AssertEquals(
    Expected := expected,
    Actual := actual,
    Message := 'Value did not update target'
);

TEST_FINISHED();
END_METHOD

METHOD PUBLIC TestSerializeTypeWith
VAR
    _type : _LINT(0);
    serializer : JsonSerializer;
    expected : STRING(500) := '{"typeName":"LINT","minValue":-9223372036854775808,"maxValue":9223372036854775807,"isSigned":true,"isFloat":false}';
    actual : STRING(500);
END_VAR
TEST('TestSerializeTypeWith');

serializer.Reset();
_type.SerializeTypeWith(serializer);
serializer.TryGetSerializedData(ADR(actual), SIZEOF(actual));

AssertEquals_STRING(
    Expected := expected,
    Actual := actual,
    Message := 'Serialization of type did not return correct string.'
);

TEST_FINISHED();
END_METHOD

METHOD PUBLIC TestSerializeWith
VAR
    _type : _LINT(32767);
    serializer : JsonSerializer;
    expected : STRING := '32767';
    actual : STRING(500);
END_VAR
TEST('TestSerializeWith');

serializer.Reset();
_type.SerializeWith(serializer);
serializer.TryGetSerializedData(ADR(actual), SIZEOF(actual));

AssertEquals_STRING(
    Expected := expected,
    Actual := actual,
    Message := 'Serialization of type data did not return correct string.'
);

TEST_FINISHED();
END_METHOD

METHOD PUBLIC TestSize
VAR
    _type : _LINT(0);
    expected : UDINT := SIZEOF(LINT);
    actual : UDINT;
END_VAR
TEST('TestSize');

actual := _type.Size;

AssertEquals_UDINT(
    Expected := Expected,
    Actual := actual,
    Message := 'Type did not return the correct size.'
);

TEST_FINISHED();
END_METHOD

METHOD PUBLIC TestTryDeserializeFrom
VAR
    deserializer : JsonDeserializer;
    feedback : DeserializerFeedback;
    json : STRING := '32767';
    _type : _LINT(0);
    expected : LINT := 32767;
    actual : LINT;
 END_VAR
TEST('TestTryDeserializeFrom');

deserializer.Reset();
deserializer.TryLoad(json);
_type.TryDeserializeFrom(Deserializer, Feedback);

actual := _type.Value;

AssertEquals(
    Expected := expected,
    Actual := actual,
    Message := 'Type did not deserialize correctly.'
);

TEST_FINISHED();
END_METHOD

METHOD PUBLIC TestTryMakeReferenceToFollowsReference
VAR
    _type : _LINT(0);
	target : _LINT(0);
    expected : LINT := 123;
    actual : LINT;
END_VAR
TEST('TestTryMakeReferenceToFollowsReference');

_type.TryMakeReferenceTo(target);
target.Value := 123;

actual := _type.Value;

AssertEquals(
    Expected := expected,
    Actual := actual,
    Message := 'Value did not follow target change'
);

TEST_FINISHED();
END_METHOD

METHOD PUBLIC TestTryMakeReferenceToUpdatesReference
VAR
    _type : _LINT(0);
	target : _LINT(0);
    expected : LINT := 123;
    actual : LINT;
END_VAR
TEST('TestTryMakeReferenceToUpdatesReference');

_type.TryMakeReferenceTo(target);
_type.Value := 123;

actual := target.Value;

AssertEquals(
    Expected := expected,
    Actual := actual,
    Message := 'Value did not update target'
);

TEST_FINISHED();
END_METHOD

METHOD PUBLIC TestTypeNameReturnsExpected
VAR
    _type : _LINT(0);
    expected : STRING := 'LINT';
    actual : STRING;
END_VAR
TEST('TestTypeNameReturnsExpected');

actual := _type.TypeName;

AssertEquals_STRING(
    Expected := expected,
    Actual := actual,
    Message := 'Type did not return correct iec type.'
);

TEST_FINISHED();
END_METHOD

METHOD PUBLIC TestValueReturnsExpectedAfterChange
VAR
    _type : _LINT(0);
    expected : LINT := 32767;
    actual : LINT;
END_VAR
TEST('TestValueReturnsExpectedAfterChange');

_type.Value := 32767;

actual := _type.Value;

AssertEquals(
    Expected := expected,
    Actual := actual,
    Message := 'Expected value not returned after change.'
);

TEST_FINISHED();
END_METHOD

METHOD PUBLIC TestValueReturnsExpectedAfterInit
VAR
    _type : _LINT(32767);
    expected : LINT := 32767;
    actual : LINT;
END_VAR
TEST('TestValueReturnsExpectedAfterInit');

actual := _type.Value;

AssertEquals(
    Expected := expected,
    Actual := actual,
    Message := 'Expected value not returned after Init.'
);

TEST_FINISHED();
END_METHOD

END_FUNCTION_BLOCK

// ---- mobject-datatypes/Tests/_REAL_TestSuite.TcPOU
FUNCTION_BLOCK _REAL_TestSuite EXTENDS TcUnit.FB_TestSuite
VAR
END_VAR

TestAddress();
TestClearReference();
TestClone();
TestTypeNameReturnsExpected();
TestIsFloat();
TestIsSigned();
TestMakeReferenceToFollowsReference();
TestMakeReferenceToUpdatesReference();
TestSize();
TestValueReturnsExpectedAfterInit();
TestValueReturnsExpectedAfterChange();
TestSerializeTypeWith();
TestSerializeWith();
TestTryDeserializeFrom();
TestTryMakeReferenceToFollowsReference();
TestTryMakeReferenceToUpdatesReference();

METHOD PUBLIC TestAddress
VAR
    _type : _REAL(0.0);
    notExpected : PVOID := 0;
    actual : PVOID;
END_VAR
TEST('TestAddress');

actual := _type.Address;

AssertFalse(
    Condition := (notExpected = actual),
    Message := 'Type did not return a valid address.'
);

TEST_FINISHED();
END_METHOD

METHOD PUBLIC TestClearReference
VAR
    _type : _REAL(0.0);
	target : REAL := 0.0;
    expected : REAL := 0.0;
    actual : REAL;
END_VAR
TEST('TestClearReference');

_type.MakeReferenceTo(target);
_type.ClearReference();
target := 123.4;

actual := _type.Value;

AssertEquals_REAL(
    Expected := expected,
    Actual := actual,
    Delta := REAL#0.001,
    Message := 'Value incorrectly followed target change'
);

TEST_FINISHED();
END_METHOD

METHOD PUBLIC TestClone
VAR
    _type : _REAL(123.4);
	clone : I_Datatype;
	isValidClone : BOOL;
	compareResult : DINT;
END_VAR
TEST('TestClone');

clone := _type.Clone();

isValidClone := clone <> 0;

IF isValidClone THEN
	compareResult := memcmp(_type.Address, clone.Address, clone.Size);
END_IF

AssertTrue(
	Condition := isValidClone,
	Message := 'Clone did not produce a clone'
);

AssertEquals_DINT(
	Expected := 0,
    Actual := compareResult,
    Message := 'Clone did not return a valid clone.'
);

clone.Dispose();

TEST_FINISHED();
END_METHOD

METHOD PUBLIC TestIsFloat
VAR
    _type : _REAL(0);
END_VAR
TEST('TestIsFloat');

AssertTrue(
	Condition := _type.IsFloat,
    Message := 'Type did not correctly identify itself as being unsigned'
);

TEST_FINISHED();
END_METHOD

METHOD PUBLIC TestIsSigned
VAR
    _type : _REAL(0);
END_VAR
TEST('TestIsSigned');

AssertTrue(
	Condition := _type.IsSigned,
    Message := 'Type did not correctly identify itself as being signed'
);

TEST_FINISHED();
END_METHOD

METHOD PUBLIC TestMakeReferenceToFollowsReference
VAR
    _type : _REAL(0.0);
	target : REAL := 0.0;
    expected : REAL := 123.4;
    actual : REAL;
END_VAR
TEST('TestMakeReferenceToFollowsReference');

_type.MakeReferenceTo(target);
target := 123.4;

actual := _type.Value;

AssertEquals_REAL(
    Expected := expected,
    Actual := actual,
    Delta := REAL#0.001,
    Message := 'Value did not follow target change'
);

TEST_FINISHED();
END_METHOD

METHOD PUBLIC TestMakeReferenceToUpdatesReference
VAR
    _type : _REAL(0.0);
	target : REAL := 0.0;
    expected : REAL := 123.4;
    actual : REAL;
END_VAR
TEST('TestMakeReferenceToUpdatesReference');

_type.MakeReferenceTo(target);
_type.Value := 123.4;

actual := target;

AssertEquals_REAL(
    Expected := expected,
    Actual := actual,
    Delta := REAL#0.001,
    Message := 'Value did not update target'
);

TEST_FINISHED();
END_METHOD

METHOD PUBLIC TestSerializeTypeWith
VAR
    _type : _REAL(0.0);
    serializer : JsonSerializer;
    expected : STRING(500) := '{"typeName":"REAL","minValue":-3.4028230607370965e38,"maxValue":3.4028230607370965e38,"isSigned":true,"isFloat":true}';
    actual : STRING(500);
END_VAR
TEST('TestSerializeTypeWith');

serializer.Reset();
_type.SerializeTypeWith(serializer);
serializer.TryGetSerializedData(ADR(actual), SIZEOF(actual));

AssertEquals_STRING(
    Expected := expected,
    Actual := actual,
    Message := 'Serialization of type did not return correct string.'
);

TEST_FINISHED();
END_METHOD

METHOD PUBLIC TestSerializeWith
VAR
    _type : _REAL(123.4);
    serializer : JsonSerializer;
    expected : STRING := '123.4000015258789'; // Expected value due to the nature of floating point values defined by IEEE754.
    actual : STRING(500);
END_VAR
TEST('TestSerializeWith');

serializer.Reset();
_type.SerializeWith(serializer);
serializer.TryGetSerializedData(ADR(actual), SIZEOF(actual));

AssertEquals_STRING(
    Expected := expected,
    Actual := actual,
    Message := 'Serialization of type data did not return correct string.'
);

TEST_FINISHED();
END_METHOD

METHOD PUBLIC TestSize
VAR
    _type : _REAL(0.0);
    expected : UDINT := SIZEOF(REAL);
    actual : UDINT;
END_VAR
TEST('TestSize');

actual := _type.Size;

AssertEquals_UDINT(
    Expected := Expected,
    Actual := actual,
    Message := 'Type did not return the correct size.'
);

TEST_FINISHED();
END_METHOD

METHOD PUBLIC TestTryDeserializeFrom
VAR
    deserializer : JsonDeserializer;
    feedback : DeserializerFeedback;
    json : STRING := '123.4';
    _type : _REAL(0.0);
    expected : REAL := 123.4;
    actual : REAL;
 END_VAR
TEST('TestTryDeserializeFrom');

deserializer.Reset();
deserializer.TryLoad(json);
_type.TryDeserializeFrom(Deserializer, Feedback);

actual := _type.Value;

AssertEquals_REAL(
    Expected := expected,
    Actual := actual,
    Delta := REAL#0.001,
    Message := 'Type did not deserialize correctly.'
);

TEST_FINISHED();
END_METHOD

METHOD PUBLIC TestTryMakeReferenceToFollowsReference
VAR
    _type : _REAL(0.0);
	target : _REAL(0.0);
    expected : REAL := 123.4;
    actual : REAL;
END_VAR
TEST('TestTryMakeReferenceToFollowsReference');

_type.TryMakeReferenceTo(target);
target.Value := 123.4;

actual := _type.Value;

AssertEquals_REAL(
    Expected := expected,
    Actual := actual,
    Delta := REAL#0.001,
    Message := 'Value did not follow target change'
);

TEST_FINISHED();
END_METHOD

METHOD PUBLIC TestTryMakeReferenceToUpdatesReference
VAR
    _type : _REAL(0.0);
	target : _REAL(0.0);
    expected : REAL := 123.4;
    actual : REAL;
END_VAR
TEST('TestTryMakeReferenceToUpdatesReference');

_type.TryMakeReferenceTo(target);
_type.Value := 123.4;

actual := target.Value;

AssertEquals_REAL(
    Expected := expected,
    Actual := actual,
    Delta := REAL#0.001,
    Message := 'Value did not update target'
);

TEST_FINISHED();
END_METHOD

METHOD PUBLIC TestTypeNameReturnsExpected
VAR
    _type : _REAL(0.0);
    expected : STRING := 'REAL';
    actual : STRING;
END_VAR
TEST('TestTypeNameReturnsExpected');

actual := _type.TypeName;

AssertEquals_STRING(
    Expected := expected,
    Actual := actual,
    Message := 'Type did not return correct iec type.'
);

TEST_FINISHED();
END_METHOD

METHOD PUBLIC TestValueReturnsExpectedAfterChange
VAR
    _type : _REAL(0.0);
    expected : REAL := 123.4;
    actual : REAL;
END_VAR
TEST('TestValueReturnsExpectedAfterChange');

_type.Value := 123.4;

actual := _type.Value;

AssertEquals_REAL(
    Expected := expected,
    Actual := actual,
    Delta := REAL#0.001,
    Message := 'Expected value not returned after change.'
);

TEST_FINISHED();
END_METHOD

METHOD PUBLIC TestValueReturnsExpectedAfterInit
VAR
    _type : _REAL(123.4);
    expected : REAL := 123.4;
    actual : REAL;
END_VAR
TEST('TestValueReturnsExpectedAfterInit');

actual := _type.Value;

AssertEquals_REAL(
    Expected := expected,
    Actual := actual,
    Delta := REAL#0.001,
    Message := 'Expected value not returned after Init.'
);

TEST_FINISHED();
END_METHOD

END_FUNCTION_BLOCK

// ---- mobject-datatypes/Tests/_SINT_TestSuite.TcPOU
FUNCTION_BLOCK _SINT_TestSuite EXTENDS TcUnit.FB_TestSuite
VAR
END_VAR

TestAddress();
TestClearReference();
TestClone();
TestTypeNameReturnsExpected();
TestIsFloat();
TestIsSigned();
TestMakeReferenceToFollowsReference();
TestMakeReferenceToUpdatesReference();
TestSize();
TestValueReturnsExpectedAfterInit();
TestValueReturnsExpectedAfterChange();
TestSerializeTypeWith();
TestSerializeWith();
TestTryDeserializeFrom();
TestTryMakeReferenceToFollowsReference();
TestTryMakeReferenceToUpdatesReference();

METHOD PUBLIC TestAddress
VAR
    _type : _SINT(0);
    notExpected : PVOID := 0;
    actual : PVOID;
END_VAR
TEST('TestAddress');

actual := _type.Address;

AssertFalse(
    Condition := (notExpected = actual),
    Message := 'Type did not return a valid address.'
);

TEST_FINISHED();
END_METHOD

METHOD PUBLIC TestClearReference
VAR
    _type : _SINT(0);
	target : SINT := 0;
    expected : SINT := 0;
    actual : SINT;
END_VAR
TEST('TestClearReference');

_type.MakeReferenceTo(target);
_type.ClearReference();
target := 123;

actual := _type.Value;

AssertEquals(
    Expected := expected,
    Actual := actual,
    Message := 'Value incorrectly followed target change'
);

TEST_FINISHED();
END_METHOD

METHOD PUBLIC TestClone
VAR
    _type : _SINT(123);
	clone : I_Datatype;
	isValidClone : BOOL;
	compareResult : DINT;
END_VAR
TEST('TestClone');

clone := _type.Clone();

isValidClone := clone <> 0;

IF isValidClone THEN
	compareResult := memcmp(_type.Address, clone.Address, clone.Size);
END_IF

AssertTrue(
	Condition := isValidClone,
	Message := 'Clone did not produce a clone'
);

AssertEquals_DINT(
	Expected := 0,
    Actual := compareResult,
    Message := 'Clone did not return a valid clone.'
);

clone.Dispose();

TEST_FINISHED();
END_METHOD

METHOD PUBLIC TestIsFloat
VAR
    _type : _SINT(0);
END_VAR
TEST('TestIsFloat');

AssertFalse(
	Condition := _type.IsFloat,
    Message := 'Type did not correctly identify itself as being unsigned'
);

TEST_FINISHED();
END_METHOD

METHOD PUBLIC TestIsSigned
VAR
    _type : _SINT(0);
END_VAR
TEST('TestIsSigned');

AssertTrue(
	Condition := _type.IsSigned,
    Message := 'Type did not correctly identify itself as being signed'
);

TEST_FINISHED();
END_METHOD

METHOD PUBLIC TestMakeReferenceToFollowsReference
VAR
    _type : _SINT(0);
	target : SINT := 0;
    expected : SINT := 123;
    actual : SINT;
END_VAR
TEST('TestMakeReferenceToFollowsReference');

_type.MakeReferenceTo(target);
target := 123;

actual := _type.Value;

AssertEquals(
    Expected := expected,
    Actual := actual,
    Message := 'Value did not follow target change'
);

TEST_FINISHED();
END_METHOD

METHOD PUBLIC TestMakeReferenceToUpdatesReference
VAR
    _type : _SINT(0);
	target : SINT := 0;
    expected : SINT := 123;
    actual : SINT;
END_VAR
TEST('TestMakeReferenceToUpdatesReference');

_type.MakeReferenceTo(target);
_type.Value := 123;

actual := target;

AssertEquals(
    Expected := expected,
    Actual := actual,
    Message := 'Value did not update target'
);

TEST_FINISHED();
END_METHOD

METHOD PUBLIC TestSerializeTypeWith
VAR
    _type : _SINT(0);
    serializer : JsonSerializer;
    expected : STRING(500) := '{"typeName":"SINT","minValue":-128,"maxValue":127,"isSigned":true,"isFloat":false}';
    actual : STRING(500);
END_VAR
TEST('TestSerializeTypeWith');

serializer.Reset();
_type.SerializeTypeWith(serializer);
serializer.TryGetSerializedData(ADR(actual), SIZEOF(actual));

AssertEquals_STRING(
    Expected := expected,
    Actual := actual,
    Message := 'Serialization of type did not return correct string.'
);

TEST_FINISHED();
END_METHOD

METHOD PUBLIC TestSerializeWith
VAR
    _type : _SINT(123);
    serializer : JsonSerializer;
    expected : STRING := '123';
    actual : STRING(500);
END_VAR
TEST('TestSerializeWith');

serializer.Reset();
_type.SerializeWith(serializer);
serializer.TryGetSerializedData(ADR(actual), SIZEOF(actual));

AssertEquals_STRING(
    Expected := expected,
    Actual := actual,
    Message := 'Serialization of type data did not return correct string.'
);

TEST_FINISHED();
END_METHOD

METHOD PUBLIC TestSize
VAR
    _type : _SINT(0);
    expected : UDINT := SIZEOF(SINT);
    actual : UDINT;
END_VAR
TEST('TestSize');

actual := _type.Size;

AssertEquals_UDINT(
    Expected := Expected,
    Actual := actual,
    Message := 'Type did not return the correct size.'
);

TEST_FINISHED();
END_METHOD

METHOD PUBLIC TestTryDeserializeFrom
VAR
    deserializer : JsonDeserializer;
    feedback : DeserializerFeedback;
    json : STRING := '123';
    _type : _SINT(0);
    expected : SINT := 123;
    actual : SINT;
 END_VAR
TEST('TestTryDeserializeFrom');

deserializer.Reset();
deserializer.TryLoad(json);
_type.TryDeserializeFrom(Deserializer, Feedback);

actual := _type.Value;

AssertEquals(
    Expected := expected,
    Actual := actual,
    Message := 'Type did not deserialize correctly.'
);

TEST_FINISHED();
END_METHOD

METHOD PUBLIC TestTryMakeReferenceToFollowsReference
VAR
    _type : _SINT(0);
	target : _SINT(0);
    expected : SINT := 123;
    actual : SINT;
END_VAR
TEST('TestTryMakeReferenceToFollowsReference');

_type.TryMakeReferenceTo(target);
target.Value := 123;

actual := _type.Value;

AssertEquals(
    Expected := expected,
    Actual := actual,
    Message := 'Value did not follow target change'
);

TEST_FINISHED();
END_METHOD

METHOD PUBLIC TestTryMakeReferenceToUpdatesReference
VAR
    _type : _SINT(0);
	target : _SINT(0);
    expected : SINT := 123;
    actual : SINT;
END_VAR
TEST('TestTryMakeReferenceToUpdatesReference');

_type.TryMakeReferenceTo(target);
_type.Value := 123;

actual := target.Value;

AssertEquals(
    Expected := expected,
    Actual := actual,
    Message := 'Value did not update target'
);

TEST_FINISHED();
END_METHOD

METHOD PUBLIC TestTypeNameReturnsExpected
VAR
    _type : _SINT(0);
    expected : STRING := 'SINT';
    actual : STRING;
END_VAR
TEST('TestTypeNameReturnsExpected');

actual := _type.TypeName;

AssertEquals_STRING(
    Expected := expected,
    Actual := actual,
    Message := 'Type did not return correct iec type.'
);

TEST_FINISHED();
END_METHOD

METHOD PUBLIC TestValueReturnsExpectedAfterChange
VAR
    _type : _SINT(0);
    expected : SINT := 123;
    actual : SINT;
END_VAR
TEST('TestValueReturnsExpectedAfterChange');

_type.Value := 123;

actual := _type.Value;

AssertEquals(
    Expected := expected,
    Actual := actual,
    Message := 'Expected value not returned after change.'
);

TEST_FINISHED();
END_METHOD

METHOD PUBLIC TestValueReturnsExpectedAfterInit
VAR
    _type : _SINT(123);
    expected : SINT := 123;
    actual : SINT;
END_VAR
TEST('TestValueReturnsExpectedAfterInit');

actual := _type.Value;

AssertEquals(
    Expected := expected,
    Actual := actual,
    Message := 'Expected value not returned after Init.'
);

TEST_FINISHED();
END_METHOD

END_FUNCTION_BLOCK

// ---- mobject-datatypes/Tests/_UDINT_TestSuite.TcPOU
FUNCTION_BLOCK _UDINT_TestSuite EXTENDS TcUnit.FB_TestSuite
VAR
END_VAR

TestAddress();
TestClearReference();
TestClone();
TestTypeNameReturnsExpected();
TestIsFloat();
TestIsSigned();
TestMakeReferenceToFollowsReference();
TestMakeReferenceToUpdatesReference();
TestSize();
TestValueReturnsExpectedAfterInit();
TestValueReturnsExpectedAfterChange();
TestSerializeTypeWith();
TestSerializeWith();
TestTryDeserializeFrom();
TestTryMakeReferenceToFollowsReference();
TestTryMakeReferenceToUpdatesReference();

METHOD PUBLIC TestAddress
VAR
    _type : _UDINT(0);
    notExpected : PVOID := 0;
    actual : PVOID;
END_VAR
TEST('TestAddress');

actual := _type.Address;

AssertFalse(
    Condition := (notExpected = actual),
    Message := 'Type did not return a valid address.'
);

TEST_FINISHED();
END_METHOD

METHOD PUBLIC TestClearReference
VAR
    _type : _UDINT(0);
	target : UDINT := 0;
    expected : UDINT := 0;
    actual : UDINT;
END_VAR
TEST('TestClearReference');

_type.MakeReferenceTo(target);
_type.ClearReference();
target := 123;

actual := _type.Value;

AssertEquals(
    Expected := expected,
    Actual := actual,
    Message := 'Value incorrectly followed target change'
);

TEST_FINISHED();
END_METHOD

METHOD PUBLIC TestClone
VAR
    _type : _UDINT(123);
	clone : I_Datatype;
	isValidClone : BOOL;
	compareResult : DINT;
END_VAR
TEST('TestClone');

clone := _type.Clone();

isValidClone := clone <> 0;

IF isValidClone THEN
	compareResult := memcmp(_type.Address, clone.Address, clone.Size);
END_IF

AssertTrue(
	Condition := isValidClone,
	Message := 'Clone did not produce a clone'
);

AssertEquals_DINT(
	Expected := 0,
    Actual := compareResult,
    Message := 'Clone did not return a valid clone.'
);

clone.Dispose();

TEST_FINISHED();
END_METHOD

METHOD PUBLIC TestIsFloat
VAR
    _type : _UDINT(0);
END_VAR
TEST('TestIsFloat');

AssertFalse(
	Condition := _type.IsFloat,
    Message := 'Type did not correctly identify itself as being unsigned'
);

TEST_FINISHED();
END_METHOD

METHOD PUBLIC TestIsSigned
VAR
    _type : _UDINT(0);
END_VAR
TEST('TestIsSigned');

AssertFalse(
	Condition := _type.IsSigned,
    Message := 'Type did not correctly identify itself as being unsigned'
);

TEST_FINISHED();
END_METHOD

METHOD PUBLIC TestMakeReferenceToFollowsReference
VAR
    _type : _UDINT(0);
	target : UDINT := 0;
    expected : UDINT := 123;
    actual : UDINT;
END_VAR
TEST('TestMakeReferenceToFollowsReference');

_type.MakeReferenceTo(target);
target := 123;

actual := _type.Value;

AssertEquals(
    Expected := expected,
    Actual := actual,
    Message := 'Value did not follow target change'
);

TEST_FINISHED();
END_METHOD

METHOD PUBLIC TestMakeReferenceToUpdatesReference
VAR
    _type : _UDINT(0);
	target : UDINT := 0;
    expected : UDINT := 123;
    actual : UDINT;
END_VAR
TEST('TestMakeReferenceToUpdatesReference');

_type.MakeReferenceTo(target);
_type.Value := 123;

actual := target;

AssertEquals(
    Expected := expected,
    Actual := actual,
    Message := 'Value did not update target'
);

TEST_FINISHED();
END_METHOD

METHOD PUBLIC TestSerializeTypeWith
VAR
    _type : _UDINT(0);
    serializer : JsonSerializer;
    expected : STRING(500) := '{"typeName":"UDINT","minValue":0,"maxValue":4294967295,"isSigned":false,"isFloat":false}';
    actual : STRING(500);
END_VAR
TEST('TestSerializeTypeWith');

serializer.Reset();
_type.SerializeTypeWith(serializer);
serializer.TryGetSerializedData(ADR(actual), SIZEOF(actual));

AssertEquals_STRING(
    Expected := expected,
    Actual := actual,
    Message := 'Serialization of type did not return correct string.'
);

TEST_FINISHED();
END_METHOD

METHOD PUBLIC TestSerializeWith
VAR
    _type : _UDINT(123);
    serializer : JsonSerializer;
    expected : STRING := '123';
    actual : STRING(500);
END_VAR
TEST('TestSerializeWith');

serializer.Reset();
_type.SerializeWith(serializer);
serializer.TryGetSerializedData(ADR(actual), SIZEOF(actual));

AssertEquals_STRING(
    Expected := expected,
    Actual := actual,
    Message := 'Serialization of type data did not return correct string.'
);

TEST_FINISHED();
END_METHOD

METHOD PUBLIC TestSize
VAR
    _type : _UDINT(0);
    expected : UDINT := SIZEOF(UDINT);
    actual : UDINT;
END_VAR
TEST('TestSize');

actual := _type.Size;

AssertEquals_UDINT(
    Expected := Expected,
    Actual := actual,
    Message := 'Type did not return the correct size.'
);

TEST_FINISHED();
END_METHOD

METHOD PUBLIC TestTryDeserializeFrom
VAR
    deserializer : JsonDeserializer;
    feedback : DeserializerFeedback;
    json : STRING := '123';
    _type : _UDINT(0);
    expected : UDINT := 123;
    actual : UDINT;
 END_VAR
TEST('TestTryDeserializeFrom');

deserializer.Reset();
deserializer.TryLoad(json);
_type.TryDeserializeFrom(Deserializer, Feedback);

actual := _type.Value;

AssertEquals(
    Expected := expected,
    Actual := actual,
    Message := 'Type did not deserialize correctly.'
);

TEST_FINISHED();
END_METHOD

METHOD PUBLIC TestTryMakeReferenceToFollowsReference
VAR
    _type : _UDINT(0);
	target : _UDINT(0);
    expected : UDINT := 123;
    actual : UDINT;
END_VAR
TEST('TestTryMakeReferenceToFollowsReference');

_type.TryMakeReferenceTo(target);
target.Value := 123;

actual := _type.Value;

AssertEquals(
    Expected := expected,
    Actual := actual,
    Message := 'Value did not follow target change'
);

TEST_FINISHED();
END_METHOD

METHOD PUBLIC TestTryMakeReferenceToUpdatesReference
VAR
    _type : _UDINT(0);
	target : _UDINT(0);
    expected : UDINT := 123;
    actual : UDINT;
END_VAR
TEST('TestTryMakeReferenceToUpdatesReference');

_type.TryMakeReferenceTo(target);
_type.Value := 123;

actual := target.Value;

AssertEquals(
    Expected := expected,
    Actual := actual,
    Message := 'Value did not update target'
);

TEST_FINISHED();
END_METHOD

METHOD PUBLIC TestTypeNameReturnsExpected
VAR
    _type : _UDINT(0);
    expected : STRING := 'UDINT';
    actual : STRING;
END_VAR
TEST('TestTypeNameReturnsExpected');

actual := _type.TypeName;

AssertEquals_STRING(
    Expected := expected,
    Actual := actual,
    Message := 'Type did not return correct iec type.'
);

TEST_FINISHED();
END_METHOD

METHOD PUBLIC TestValueReturnsExpectedAfterChange
VAR
    _type : _UDINT(0);
    expected : UDINT := 123;
    actual : UDINT;
END_VAR
TEST('TestValueReturnsExpectedAfterChange');

_type.Value := 123;

actual := _type.Value;

AssertEquals(
    Expected := expected,
    Actual := actual,
    Message := 'Expected value not returned after change.'
);

TEST_FINISHED();
END_METHOD

METHOD PUBLIC TestValueReturnsExpectedAfterInit
VAR
    _type : _UDINT(123);
    expected : UDINT := 123;
    actual : UDINT;
END_VAR
TEST('TestValueReturnsExpectedAfterInit');

actual := _type.Value;

AssertEquals(
    Expected := expected,
    Actual := actual,
    Message := 'Expected value not returned after Init.'
);

TEST_FINISHED();
END_METHOD

END_FUNCTION_BLOCK

// ---- mobject-datatypes/Tests/_UINT_TestSuite.TcPOU
FUNCTION_BLOCK _UINT_TestSuite EXTENDS TcUnit.FB_TestSuite
VAR
END_VAR

TestAddress();
TestClearReference();
TestClone();
TestTypeNameReturnsExpected();
TestIsFloat();
TestIsSigned();
TestMakeReferenceToFollowsReference();
TestMakeReferenceToUpdatesReference();
TestSize();
TestValueReturnsExpectedAfterInit();
TestValueReturnsExpectedAfterChange();
TestSerializeTypeWith();
TestSerializeWith();
TestTryDeserializeFrom();
TestTryMakeReferenceToFollowsReference();
TestTryMakeReferenceToUpdatesReference();

METHOD PUBLIC TestAddress
VAR
    _type : _UINT(0);
    notExpected : PVOID := 0;
    actual : PVOID;
END_VAR
TEST('TestAddress');

actual := _type.Address;

AssertFalse(
    Condition := (notExpected = actual),
    Message := 'Type did not return a valid address.'
);

TEST_FINISHED();
END_METHOD

METHOD PUBLIC TestClearReference
VAR
    _type : _UINT(0);
	target : UINT := 0;
    expected : UINT := 0;
    actual : UINT;
END_VAR
TEST('TestClearReference');

_type.MakeReferenceTo(target);
_type.ClearReference();
target := 123;

actual := _type.Value;

AssertEquals(
    Expected := expected,
    Actual := actual,
    Message := 'Value incorrectly followed target change'
);

TEST_FINISHED();
END_METHOD

METHOD PUBLIC TestClone
VAR
    _type : _UINT(123);
	clone : I_Datatype;
	isValidClone : BOOL;
	compareResult : DINT;
END_VAR
TEST('TestClone');

clone := _type.Clone();

isValidClone := clone <> 0;

IF isValidClone THEN
	compareResult := memcmp(_type.Address, clone.Address, clone.Size);
END_IF

AssertTrue(
	Condition := isValidClone,
	Message := 'Clone did not produce a clone'
);

AssertEquals_DINT(
	Expected := 0,
    Actual := compareResult,
    Message := 'Clone did not return a valid clone.'
);

clone.Dispose();

TEST_FINISHED();
END_METHOD

METHOD PUBLIC TestIsFloat
VAR
    _type : _UINT(0);
END_VAR
TEST('TestIsFloat');

AssertFalse(
	Condition := _type.IsFloat,
    Message := 'Type did not correctly identify itself as being unsigned'
);

TEST_FINISHED();
END_METHOD

METHOD PUBLIC TestIsSigned
VAR
    _type : _UINT(0);
END_VAR
TEST('TestIsSigned');

AssertFalse(
	Condition := _type.IsSigned,
    Message := 'Type did not correctly identify itself as being unsigned'
);

TEST_FINISHED();
END_METHOD

METHOD PUBLIC TestMakeReferenceToFollowsReference
VAR
    _type : _UINT(0);
	target : UINT := 0;
    expected : UINT := 123;
    actual : UINT;
END_VAR
TEST('TestMakeReferenceToFollowsReference');

_type.MakeReferenceTo(target);
target := 123;

actual := _type.Value;

AssertEquals(
    Expected := expected,
    Actual := actual,
    Message := 'Value did not follow target change'
);

TEST_FINISHED();
END_METHOD

METHOD PUBLIC TestMakeReferenceToUpdatesReference
VAR
    _type : _UINT(0);
	target : UINT := 0;
    expected : UINT := 123;
    actual : UINT;
END_VAR
TEST('TestMakeReferenceToUpdatesReference');

_type.MakeReferenceTo(target);
_type.Value := 123;

actual := target;

AssertEquals(
    Expected := expected,
    Actual := actual,
    Message := 'Value did not update target'
);

TEST_FINISHED();
END_METHOD

METHOD PUBLIC TestSerializeTypeWith
VAR
    _type : _UINT(0);
    serializer : JsonSerializer;
    expected : STRING(500) := '{"typeName":"UINT","minValue":0,"maxValue":65535,"isSigned":false,"isFloat":false}';
    actual : STRING(500);
END_VAR
TEST('TestSerializeTypeWith');

serializer.Reset();
_type.SerializeTypeWith(serializer);
serializer.TryGetSerializedData(ADR(actual), SIZEOF(actual));

AssertEquals_STRING(
    Expected := expected,
    Actual := actual,
    Message := 'Serialization of type did not return correct string.'
);

TEST_FINISHED();
END_METHOD

METHOD PUBLIC TestSerializeWith
VAR
    _type : _UINT(123);
    serializer : JsonSerializer;
    expected : STRING := '123';
    actual : STRING(500);
END_VAR
TEST('TestSerializeWith');

serializer.Reset();
_type.SerializeWith(serializer);
serializer.TryGetSerializedData(ADR(actual), SIZEOF(actual));

AssertEquals_STRING(
    Expected := expected,
    Actual := actual,
    Message := 'Serialization of type data did not return correct string.'
);

TEST_FINISHED();
END_METHOD

METHOD PUBLIC TestSize
VAR
    _type : _UINT(0);
    expected : UDINT := SIZEOF(UINT);
    actual : UDINT;
END_VAR
TEST('TestSize');

actual := _type.Size;

AssertEquals_UDINT(
    Expected := Expected,
    Actual := actual,
    Message := 'Type did not return the correct size.'
);

TEST_FINISHED();
END_METHOD

METHOD PUBLIC TestTryDeserializeFrom
VAR
    deserializer : JsonDeserializer;
    feedback : DeserializerFeedback;
    json : STRING := '123';
    _type : _UINT(0);
    expected : UINT := 123;
    actual : UINT;
 END_VAR
TEST('TestTryDeserializeFrom');

deserializer.Reset();
deserializer.TryLoad(json);
_type.TryDeserializeFrom(Deserializer, Feedback);

actual := _type.Value;

AssertEquals(
    Expected := expected,
    Actual := actual,
    Message := 'Type did not deserialize correctly.'
);

TEST_FINISHED();
END_METHOD

METHOD PUBLIC TestTryMakeReferenceToFollowsReference
VAR
    _type : _UINT(0);
	target : _UINT(0);
    expected : UINT := 123;
    actual : UINT;
END_VAR
TEST('TestTryMakeReferenceToFollowsReference');

_type.TryMakeReferenceTo(target);
target.Value := 123;

actual := _type.Value;

AssertEquals(
    Expected := expected,
    Actual := actual,
    Message := 'Value did not follow target change'
);

TEST_FINISHED();
END_METHOD

METHOD PUBLIC TestTryMakeReferenceToUpdatesReference
VAR
    _type : _UINT(0);
	target : _UINT(0);
    expected : UINT := 123;
    actual : UINT;
END_VAR
TEST('TestTryMakeReferenceToUpdatesReference');

_type.TryMakeReferenceTo(target);
_type.Value := 123;

actual := target.Value;

AssertEquals(
    Expected := expected,
    Actual := actual,
    Message := 'Value did not update target'
);

TEST_FINISHED();
END_METHOD

METHOD PUBLIC TestTypeNameReturnsExpected
VAR
    _type : _UINT(0);
    expected : STRING := 'UINT';
    actual : STRING;
END_VAR
TEST('TestTypeNameReturnsExpected');

actual := _type.TypeName;

AssertEquals_STRING(
    Expected := expected,
    Actual := actual,
    Message := 'Type did not return correct iec type.'
);

TEST_FINISHED();
END_METHOD

METHOD PUBLIC TestValueReturnsExpectedAfterChange
VAR
    _type : _UINT(0);
    expected : UINT := 123;
    actual : UINT;
END_VAR
TEST('TestValueReturnsExpectedAfterChange');

_type.Value := 123;

actual := _type.Value;

AssertEquals(
    Expected := expected,
    Actual := actual,
    Message := 'Expected value not returned after change.'
);

TEST_FINISHED();
END_METHOD

METHOD PUBLIC TestValueReturnsExpectedAfterInit
VAR
    _type : _UINT(123);
    expected : UINT := 123;
    actual : UINT;
END_VAR
TEST('TestValueReturnsExpectedAfterInit');

actual := _type.Value;

AssertEquals(
    Expected := expected,
    Actual := actual,
    Message := 'Expected value not returned after Init.'
);

TEST_FINISHED();
END_METHOD

END_FUNCTION_BLOCK

// ---- mobject-datatypes/Tests/_ULINT_TestSuite.TcPOU
FUNCTION_BLOCK _ULINT_TestSuite EXTENDS TcUnit.FB_TestSuite
VAR
END_VAR

TestAddress();
TestClearReference();
TestClone();
TestTypeNameReturnsExpected();
TestIsFloat();
TestIsSigned();
TestMakeReferenceToFollowsReference();
TestMakeReferenceToUpdatesReference();
TestSize();
TestValueReturnsExpectedAfterInit();
TestValueReturnsExpectedAfterChange();
TestSerializeTypeWith();
TestSerializeWith();
TestTryDeserializeFrom();
TestTryMakeReferenceToFollowsReference();
TestTryMakeReferenceToUpdatesReference();

METHOD PUBLIC TestAddress
VAR
    _type : _ULINT(0);
    notExpected : PVOID := 0;
    actual : PVOID;
END_VAR
TEST('TestAddress');

actual := _type.Address;

AssertFalse(
    Condition := (notExpected = actual),
    Message := 'Type did not return a valid address.'
);

TEST_FINISHED();
END_METHOD

METHOD PUBLIC TestClearReference
VAR
    _type : _ULINT(0);
	target : ULINT := 0;
    expected : ULINT := 0;
    actual : ULINT;
END_VAR
TEST('TestClearReference');

_type.MakeReferenceTo(target);
_type.ClearReference();
target := 123;

actual := _type.Value;

AssertEquals(
    Expected := expected,
    Actual := actual,
    Message := 'Value incorrectly followed target change'
);

TEST_FINISHED();
END_METHOD

METHOD PUBLIC TestClone
VAR
    _type : _ULINT(123);
	clone : I_Datatype;
	isValidClone : BOOL;
	compareResult : DINT;
END_VAR
TEST('TestClone');

clone := _type.Clone();

isValidClone := clone <> 0;

IF isValidClone THEN
	compareResult := memcmp(_type.Address, clone.Address, clone.Size);
END_IF

AssertTrue(
	Condition := isValidClone,
	Message := 'Clone did not produce a clone'
);

AssertEquals_DINT(
	Expected := 0,
    Actual := compareResult,
    Message := 'Clone did not return a valid clone.'
);

clone.Dispose();

TEST_FINISHED();
END_METHOD

METHOD PUBLIC TestIsFloat
VAR
    _type : _ULINT(0);
END_VAR
TEST('TestIsFloat');

AssertFalse(
	Condition := _type.IsFloat,
    Message := 'Type did not correctly identify itself as being unsigned'
);

TEST_FINISHED();
END_METHOD

METHOD PUBLIC TestIsSigned
VAR
    _type : _ULINT(0);
END_VAR
TEST('TestIsSigned');

AssertFalse(
	Condition := _type.IsSigned,
    Message := 'Type did not correctly identify itself as being unsigned'
);

TEST_FINISHED();
END_METHOD

METHOD PUBLIC TestMakeReferenceToFollowsReference
VAR
    _type : _ULINT(0);
	target : ULINT := 0;
    expected : ULINT := 123;
    actual : ULINT;
END_VAR
TEST('TestMakeReferenceToFollowsReference');

_type.MakeReferenceTo(target);
target := 123;

actual := _type.Value;

AssertEquals(
    Expected := expected,
    Actual := actual,
    Message := 'Value did not follow target change'
);

TEST_FINISHED();
END_METHOD

METHOD PUBLIC TestMakeReferenceToUpdatesReference
VAR
    _type : _ULINT(0);
	target : ULINT := 0;
    expected : ULINT := 123;
    actual : ULINT;
END_VAR
TEST('TestMakeReferenceToUpdatesReference');

_type.MakeReferenceTo(target);
_type.Value := 123;

actual := target;

AssertEquals(
    Expected := expected,
    Actual := actual,
    Message := 'Value did not update target'
);

TEST_FINISHED();
END_METHOD

METHOD PUBLIC TestSerializeTypeWith
VAR
    _type : _ULINT(0);
    serializer : JsonSerializer;
    expected : STRING(500) := '{"typeName":"ULINT","minValue":0,"maxValue":18446744073709551615,"isSigned":false,"isFloat":false}';
    actual : STRING(500);
END_VAR
TEST('TestSerializeTypeWith');

serializer.Reset();
_type.SerializeTypeWith(serializer);
serializer.TryGetSerializedData(ADR(actual), SIZEOF(actual));

AssertEquals_STRING(
    Expected := expected,
    Actual := actual,
    Message := 'Serialization of type did not return correct string.'
);

TEST_FINISHED();
END_METHOD

METHOD PUBLIC TestSerializeWith
VAR
    _type : _ULINT(32767);
    serializer : JsonSerializer;
    expected : STRING := '32767';
    actual : STRING(500);
END_VAR
TEST('TestSerializeWith');

serializer.Reset();
_type.SerializeWith(serializer);
serializer.TryGetSerializedData(ADR(actual), SIZEOF(actual));

AssertEquals_STRING(
    Expected := expected,
    Actual := actual,
    Message := 'Serialization of type data did not return correct string.'
);

TEST_FINISHED();
END_METHOD

METHOD PUBLIC TestSize
VAR
    _type : _ULINT(0);
    expected : UDINT := SIZEOF(ULINT);
    actual : UDINT;
END_VAR
TEST('TestSize');

actual := _type.Size;

AssertEquals_UDINT(
    Expected := Expected,
    Actual := actual,
    Message := 'Type did not return the correct size.'
);

TEST_FINISHED();
END_METHOD

METHOD PUBLIC TestTryDeserializeFrom
VAR
    deserializer : JsonDeserializer;
    feedback : DeserializerFeedback;
    json : STRING := '32767';
    _type : _ULINT(0);
    expected : ULINT := 32767;
    actual : ULINT;
 END_VAR
TEST('TestTryDeserializeFrom');

deserializer.Reset();
deserializer.TryLoad(json);
_type.TryDeserializeFrom(Deserializer, Feedback);

actual := _type.Value;

AssertEquals(
    Expected := expected,
    Actual := actual,
    Message := 'Type did not deserialize correctly.'
);

TEST_FINISHED();
END_METHOD

METHOD PUBLIC TestTryMakeReferenceToFollowsReference
VAR
    _type : _ULINT(0);
	target : _ULINT(0);
    expected : ULINT := 123;
    actual : ULINT;
END_VAR
TEST('TestTryMakeReferenceToFollowsReference');

_type.TryMakeReferenceTo(target);
target.Value := 123;

actual := _type.Value;

AssertEquals(
    Expected := expected,
    Actual := actual,
    Message := 'Value did not follow target change'
);

TEST_FINISHED();
END_METHOD

METHOD PUBLIC TestTryMakeReferenceToUpdatesReference
VAR
    _type : _ULINT(0);
	target : _ULINT(0);
    expected : ULINT := 123;
    actual : ULINT;
END_VAR
TEST('TestTryMakeReferenceToUpdatesReference');

_type.TryMakeReferenceTo(target);
_type.Value := 123;

actual := target.Value;

AssertEquals(
    Expected := expected,
    Actual := actual,
    Message := 'Value did not update target'
);

TEST_FINISHED();
END_METHOD

METHOD PUBLIC TestTypeNameReturnsExpected
VAR
    _type : _ULINT(0);
    expected : STRING := 'ULINT';
    actual : STRING;
END_VAR
TEST('TestTypeNameReturnsExpected');

actual := _type.TypeName;

AssertEquals_STRING(
    Expected := expected,
    Actual := actual,
    Message := 'Type did not return correct iec type.'
);

TEST_FINISHED();
END_METHOD

METHOD PUBLIC TestValueReturnsExpectedAfterChange
VAR
    _type : _ULINT(0);
    expected : ULINT := 32767;
    actual : ULINT;
END_VAR
TEST('TestValueReturnsExpectedAfterChange');

_type.Value := 32767;

actual := _type.Value;

AssertEquals(
    Expected := expected,
    Actual := actual,
    Message := 'Expected value not returned after change.'
);

TEST_FINISHED();
END_METHOD

METHOD PUBLIC TestValueReturnsExpectedAfterInit
VAR
    _type : _ULINT(32767);
    expected : ULINT := 32767;
    actual : ULINT;
END_VAR
TEST('TestValueReturnsExpectedAfterInit');

actual := _type.Value;

AssertEquals(
    Expected := expected,
    Actual := actual,
    Message := 'Expected value not returned after Init.'
);

TEST_FINISHED();
END_METHOD

END_FUNCTION_BLOCK

// ---- mobject-deserialization/Tests/CustomDeserializationFailedError_TestSuite.TcPOU
FUNCTION_BLOCK CustomDeserializationFailedError_TestSuite EXTENDS TcUnit.FB_TestSuite

TestAccept();
TestErrorType();
TestIsSameAsWithSameErrors();
TestIsSameAsWithDifferentErrors();
TestMessage();
TestSerializeWith();

METHOD PUBLIC TestAccept
VAR
	error : CustomDeserializationFailedError(Message := 'TestMessage');
	visitor : MockErrorVisitor(ExpectedError := error);
END_VAR
TEST('TestAccept');

error.Accept(visitor);

AssertTrue(
	Condition := visitor.VisitedCorrectError,
	Message := 'Did not invoke VisitError on the visitor'
);

TEST_FINISHED();
END_METHOD

METHOD PUBLIC TestErrorType
VAR
	error : CustomDeserializationFailedError(Message := 'TestMessage');
END_VAR
TEST('TestErrorType');

AssertEquals_String(
	Actual := error.ErrorType,
	Expected := 'CUSTOM_DESERIALIZATION_ERROR',
	Message := 'Did not return the expected ErrorType'
);

TEST_FINISHED();
END_METHOD

METHOD PUBLIC TestIsSameAsWithDifferentErrors
VAR
	error1 : CustomDeserializationFailedError(Message := 'TestMessage');
	error2 : MockError(MockErrorType:='ERROR_TYPE_B',MockMessage:='TestMessage');
END_VAR
TEST('TestIsSameAsWithDifferentErrors');

AssertFalse(
	Condition := error1.IsSameAs(error2),
	Message := 'Did not correctly identify errors as being different type'
);

TEST_FINISHED();
END_METHOD

METHOD PUBLIC TestIsSameAsWithSameErrors
VAR
	error1 : CustomDeserializationFailedError(Message := 'TestMessage');
	error2 : MockError(MockErrorType:='CUSTOM_DESERIALIZATION_ERROR',MockMessage:='Deserialization Failed, TestMessage');
END_VAR
TEST('TestIsSameAsWithSameErrors');

AssertTrue(
	Condition := error1.IsSameAs(error2),
	Message := 'Did not correctly identify errors as being the same type'
);

TEST_FINISHED();
END_METHOD

METHOD PUBLIC TestMessage
VAR
	error : CustomDeserializationFailedError(Message := 'TestMessage');
END_VAR
TEST('TestMessage');

AssertEquals_String(
	Actual := error.Message,
	Expected := 'Deserialization Failed, TestMessage',
	Message := 'Did not return the expected Message'
);

TEST_FINISHED();
END_METHOD

METHOD PUBLIC TestSerializeWith
VAR
	error : CustomDeserializationFailedError(Message := 'TestMessage');
	serializer : MockJsonSerializer;
	result : T_MAXSTRING;
END_VAR
TEST('TestSerializeWith');

error.SerializeWith(serializer);
serializer.TryGetSerializedData(ADR(result), SIZEOF(result));

AssertEquals_String(
	Actual := result,
	Expected := '{"errorType":"CUSTOM_DESERIALIZATION_ERROR","message":"Deserialization Failed, TestMessage"}',
	Message := 'Did not serialize correctly'
);

TEST_FINISHED();
END_METHOD

END_FUNCTION_BLOCK

// ---- SharedMocks/MockError.TcPOU
FUNCTION_BLOCK MockError EXTENDS Error
VAR
	_errorType : T_MAXSTRING;
	_message : T_MAXSTRING;
END_VAR

PROPERTY PUBLIC ErrorType : T_MAXSTRING
GET
ErrorType := _errorType;
END_GET
END_PROPERTY

METHOD FB_init : BOOL
VAR_INPUT
	bInitRetains : BOOL; // if TRUE, the retain variables are initialized (warm start / cold start)
	bInCopyCode : BOOL;  // if TRUE, the instance afterwards gets moved into the copy code (online change)
	MockErrorType : T_MAXSTRING;
	MockMessage : T_MAXSTRING;
END_VAR
_errorType := MockErrorType;
_message := MockMessage;
END_METHOD

PROPERTY PUBLIC Message : T_MAXSTRING
GET
Message := _message;
END_GET
END_PROPERTY

END_FUNCTION_BLOCK

// ---- SharedMocks/MockJsonSerializer.TcPOU
{attribute 'linkalways'} 
{attribute 'no_explicit_call' := 'This FB is a CLASS and must be accessed using methods or properties'}
{attribute 'enable_dynamic_creation'}
// this code has been taken from mobject-json to prevent circular referencing 
FUNCTION_BLOCK MockJsonSerializer EXTENDS Disposable IMPLEMENTS I_Serializer;
VAR
	jsonSaxWriter : FB_JsonSaxWriter;
END_VAR

METHOD PUBLIC AddBase64 : I_Serializer
VAR_INPUT
	pBytes : POINTER TO BYTE;
	nBytes : DINT;
END_VAR
jsonSaxWriter.AddBase64(pBytes, nBytes);
AddBase64 := THIS^;
END_METHOD

METHOD PUBLIC AddBool : I_Serializer
VAR_INPUT
	Value : BOOL;
END_VAR
jsonSaxWriter.AddBool(Value);
AddBool := THIS^;
END_METHOD

METHOD PUBLIC AddByte : I_Serializer
VAR_INPUT
	Value : BYTE;
END_VAR
jsonSaxWriter.AddUDint(BYTE_TO_UDINT(Value));
AddByte := THIS^;
END_METHOD

METHOD PUBLIC AddBytesAsHex : I_Serializer
VAR_INPUT
	pBytes : POINTER TO BYTE;
	nBytes : DINT;
END_VAR
jsonSaxWriter.AddHexBinary(pBytes, nBytes);
AddBytesAsHex := THIS^;
END_METHOD

METHOD PUBLIC AddDateTime : I_Serializer
VAR_INPUT
	Value : DATE_AND_TIME;
END_VAR
jsonSaxWriter.AddDateTime(Value);
AddDateTime := THIS^;
END_METHOD

METHOD PUBLIC AddDcTime : I_Serializer
VAR_INPUT
	Value : DCTIME;
END_VAR
jsonSaxWriter.AddDcTime(Value);
AddDcTime := THIS^;
END_METHOD

METHOD PUBLIC AddDint : I_Serializer
VAR_INPUT
	Value : DINT;
END_VAR
jsonSaxWriter.AddDint(Value);
AddDint := THIS^;
END_METHOD

METHOD PUBLIC AddDword : I_Serializer
VAR_INPUT
	Value : DWORD;
END_VAR
jsonSaxWriter.AddUDint(DWORD_TO_UDINT(Value));
AddDword := THIS^;
END_METHOD

METHOD PUBLIC AddFileTime : I_Serializer
VAR_INPUT
	Value : FILETIME;
END_VAR
jsonSaxWriter.AddFileTime(Value);
AddFileTime := THIS^;
END_METHOD

METHOD PUBLIC AddInt : I_Serializer
VAR_INPUT
	Value : INT;
END_VAR
jsonSaxWriter.AddDint(INT_TO_DINT(Value));
AddInt := THIS^;
END_METHOD

METHOD PUBLIC AddKey : I_Serializer
VAR_INPUT
	Key : T_MAXSTRING;
END_VAR
jsonSaxWriter.AddKey(Key);
AddKey := THIS^;
END_METHOD

METHOD PUBLIC AddKeyBase64 : I_Serializer
VAR_INPUT
	Key : T_MAXSTRING;
	pBytes : POINTER TO BYTE;
	nBytes : DINT;
END_VAR
AddKey(Key);
AddBase64(pBytes, nBytes);
AddKeyBase64 := THIS^;
END_METHOD

METHOD PUBLIC AddKeyBool : I_Serializer
VAR_INPUT
	Key : T_MAXSTRING;
	Value : BOOL;
END_VAR
AddKey(Key);
AddBool(Value);
AddKeyBool := THIS^;
END_METHOD

METHOD PUBLIC AddKeyByte : I_Serializer
VAR_INPUT
	Key : T_MAXSTRING;
	Value : BYTE;
END_VAR
AddKey(Key);
AddByte(Value);
AddKeyByte := THIS^;
END_METHOD

METHOD PUBLIC AddKeyBytesAsHex : I_Serializer
VAR_INPUT
	Key : T_MAXSTRING;
	pBytes : POINTER TO BYTE;
	nBytes : DINT;
END_VAR
AddKey(Key);
AddBytesAsHex(pBytes, nBytes);
AddKeyBytesAsHex := THIS^;
END_METHOD

METHOD PUBLIC AddKeyDateTime : I_Serializer
VAR_INPUT
	Key : T_MAXSTRING;
	Value : DATE_AND_TIME;
END_VAR
AddKey(Key);
AddDateTime(Value);
AddKeyDateTime := THIS^;
END_METHOD

METHOD PUBLIC AddKeyDcTime : I_Serializer
VAR_INPUT
	Key : T_MAXSTRING;
	Value : DCTIME;
END_VAR
AddKey(Key);
AddDcTime(Value);
AddKeyDcTime := THIS^;
END_METHOD

METHOD PUBLIC AddKeyDint : I_Serializer
VAR_INPUT
	Key : T_MAXSTRING;
	Value : DINT;
END_VAR
AddKey(Key);
AddDint(Value);
AddKeyDint := THIS^;
END_METHOD

METHOD PUBLIC AddKeyDword : I_Serializer
VAR_INPUT
	Key : T_MAXSTRING;
	Value : DWORD;
END_VAR
AddKey(Key);
AddDword(Value);
AddKeyDword := THIS^;
END_METHOD

METHOD PUBLIC AddKeyFileTime : I_Serializer
VAR_INPUT
	Key : T_MAXSTRING;
	Value : FILETIME;
END_VAR
AddKey(Key);
AddFileTime(Value);
AddKeyFileTime := THIS^;
END_METHOD

METHOD PUBLIC AddKeyInt : I_Serializer
VAR_INPUT
	Key : T_MAXSTRING;
	Value : INT;
END_VAR
AddKey(Key);
AddInt(Value);
AddKeyInt := THIS^;
END_METHOD

METHOD PUBLIC AddKeyLint : I_Serializer
VAR_INPUT
	Key : T_MAXSTRING;
	Value : LINT;
END_VAR
AddKey(Key);
AddLint(Value);
AddKeyLint := THIS^;
END_METHOD

METHOD PUBLIC AddKeyLreal : I_Serializer
VAR_INPUT
	Key : T_MAXSTRING;
	Value : LREAL;
END_VAR
AddKey(Key);
AddLreal(Value);
AddKeyLreal := THIS^;
END_METHOD

METHOD PUBLIC AddKeyLtime : I_Serializer
VAR_INPUT
	Key : T_MAXSTRING;
	Value : LTIME;
END_VAR
AddKey(Key);
AddLTIME(Value);
AddKeyLtime := THIS^;
END_METHOD

METHOD PUBLIC AddKeyLword : I_Serializer
VAR_INPUT
	Key : T_MAXSTRING;
	Value : LWORD;
END_VAR
AddKey(Key);
AddLword(Value);
AddKeyLword := THIS^;
END_METHOD

METHOD PUBLIC AddKeyNull : I_Serializer
VAR_INPUT
	Key : T_MAXSTRING;
END_VAR
AddKey(Key);
AddNull();
AddKeyNull := THIS^;
END_METHOD

METHOD PUBLIC AddKeyObject : I_Serializer
VAR_INPUT
	Key : T_MAXSTRING;
	Object : I_Serializable;
END_VAR
AddKey(Key);
Object.SerializeWith(THIS^);
AddKeyObject := THIS^;
END_METHOD

METHOD PUBLIC AddKeyRawJson : I_Serializer
VAR_INPUT
	Key : T_MAXSTRING;
	RawObject : REFERENCE TO STRING;;
END_VAR
AddKey(Key);
AddRawJson(RawObject);
AddKeyRawJson := THIS^;
END_METHOD

METHOD PUBLIC AddKeyReal : I_Serializer
VAR_INPUT
	Key : T_MAXSTRING;
	Value : REAL;
END_VAR
AddKey(Key);
AddReal(Value);
AddKeyReal := THIS^;
END_METHOD

METHOD PUBLIC AddKeySint : I_Serializer
VAR_INPUT
	Key : T_MAXSTRING;
	Value : SINT;
END_VAR
AddKey(Key);
AddSint(Value);
AddKeySint := THIS^;
END_METHOD

METHOD PUBLIC AddKeyString : I_Serializer
VAR_INPUT
	Key : T_MAXSTRING;
	Value : T_MAXSTRING;
END_VAR
AddKey(Key);
AddString(Value);
AddKeyString := THIS^;
END_METHOD

METHOD PUBLIC AddKeyStringByRef : I_Serializer
VAR_INPUT
	Key : T_MAXSTRING;
	Value : REFERENCE TO STRING;;
END_VAR
AddKey(Key);
AddStringByRef(Value);
AddKeyStringByRef := THIS^;
END_METHOD

METHOD PUBLIC AddKeyTime : I_Serializer
VAR_INPUT
	Key : T_MAXSTRING;
	Value : TIME;
END_VAR
AddKey(Key);
AddTime(Value);
AddKeyTime := THIS^;
END_METHOD

METHOD PUBLIC AddKeyTod : I_Serializer
VAR_INPUT
	Key : T_MAXSTRING;
	Value : TOD;
END_VAR
AddKey(Key);
AddTod(Value);
AddKeyTod := THIS^;
END_METHOD

METHOD PUBLIC AddKeyUdint : I_Serializer
VAR_INPUT
	Key : T_MAXSTRING;
	Value : UDINT;
END_VAR
AddKey(Key);
AddUdint(Value);
AddKeyUdint := THIS^;
END_METHOD

METHOD PUBLIC AddKeyUint : I_Serializer
VAR_INPUT
	Key : T_MAXSTRING;
	Value : UINT;
END_VAR
AddKey(Key);
AddUint(Value);
AddKeyUint := THIS^;
END_METHOD

METHOD PUBLIC AddKeyUlint : I_Serializer
VAR_INPUT
	Key : T_MAXSTRING;
	Value : ULINT;
END_VAR
AddKey(Key);
AddUlint(Value);
AddKeyUlint := THIS^;
END_METHOD

METHOD PUBLIC AddKeyUsint : I_Serializer
VAR_INPUT
	Key : T_MAXSTRING;
	Value : USINT;
END_VAR
AddKey(Key);
AddUsint(Value);
AddKeyUsint := THIS^;
END_METHOD

METHOD PUBLIC AddKeyWord : I_Serializer
VAR_INPUT
	Key : T_MAXSTRING;
	Value : WORD;
END_VAR
AddKey(Key);
AddWord(Value);
AddKeyWord := THIS^;
END_METHOD

METHOD PUBLIC AddLint : I_Serializer
VAR_INPUT
	Value : LINT;
END_VAR
jsonSaxWriter.AddLint(Value);
AddLint := THIS^;
END_METHOD

METHOD PUBLIC AddLreal : I_Serializer
VAR_INPUT
	Value : LREAL;
END_VAR
jsonSaxWriter.AddLreal(Value);
AddLreal := THIS^;
END_METHOD

METHOD PUBLIC AddLtime : I_Serializer
VAR_INPUT
	Value : LTIME;
END_VAR
VAR
	converted : T_MAXSTRING;
END_VAR
converted := LTIME_TO_STRING(Value);
jsonSaxWriter.AddString(converted);
AddLtime := THIS^;
END_METHOD

METHOD PUBLIC AddLword : I_Serializer
VAR_INPUT
	Value : LWORD;
END_VAR
jsonSaxWriter.AddUlint(LWORD_TO_ULINT(Value));
AddLword := THIS^;
END_METHOD

METHOD PUBLIC AddNull : I_Serializer
VAR_INPUT
END_VAR
jsonSaxWriter.AddNull();
AddNull := THIS^;
END_METHOD

METHOD PUBLIC AddObject
VAR_INPUT
	Object : I_Serializable;
END_VAR
Object.SerializeWith(This^);
END_METHOD

METHOD PUBLIC AddRawJson
VAR_INPUT
	RawObject : REFERENCE TO STRING;
END_VAR
jsonSaxWriter.AddRawObject(RawObject);
END_METHOD

METHOD PUBLIC AddReal : I_Serializer
VAR_INPUT
	Value : REAL;
END_VAR
// real to lreal is used to negate an issue with TC4024.55 which prevents max REAL from being serailized.  
// so a REAL_TO_LREAL conversion is made to ensure this is always possible.  
jsonSaxWriter.AddLReal(REAL_TO_LREAL(Value));
AddReal := THIS^;
END_METHOD

METHOD PUBLIC AddSint : I_Serializer
VAR_INPUT
	Value : SINT;
END_VAR
jsonSaxWriter.AddDint(SINT_TO_DINT(Value));
AddSint := THIS^;
END_METHOD

METHOD PUBLIC AddString : I_Serializer
VAR_INPUT
	Value : T_MAXSTRING;
END_VAR
jsonSaxWriter.AddString(Value);
AddString := THIS^;
END_METHOD

METHOD PUBLIC AddStringByRef : I_Serializer
VAR_INPUT
	Value : REFERENCE TO STRING;
END_VAR
jsonSaxWriter.AddString(Value);
AddStringByRef := THIS^;
END_METHOD

METHOD PUBLIC AddTime : I_Serializer
VAR_INPUT
	Value : TIME;
END_VAR
VAR
	converted : T_MAXSTRING;
END_VAR
converted := TIME_TO_STRING(Value);
jsonSaxWriter.AddString(converted);
AddTime := THIS^;
END_METHOD

METHOD PUBLIC AddTod : I_Serializer
VAR_INPUT
	Value : TOD;
END_VAR
VAR
	converted : T_MAXSTRING;
END_VAR
converted := TOD_TO_STRING(Value);
jsonSaxWriter.AddString(converted);
AddTod := THIS^;
END_METHOD

METHOD PUBLIC AddUdint : I_Serializer
VAR_INPUT
	Value : UDINT;
END_VAR
jsonSaxWriter.AddUdint(Value);
AddUdint := THIS^;
END_METHOD

METHOD PUBLIC AddUint : I_Serializer
VAR_INPUT
	Value : UINT;
END_VAR
jsonSaxWriter.AddDint(UINT_TO_DINT(Value));
AddUint := THIS^;
END_METHOD

METHOD PUBLIC AddUlint : I_Serializer
VAR_INPUT
	Value : ULINT;
END_VAR
jsonSaxWriter.AddUlint(Value);
AddUlint := THIS^;
END_METHOD

METHOD PUBLIC AddUsint : I_Serializer
VAR_INPUT
	Value : USINT;
END_VAR
jsonSaxWriter.AddDint(USINT_TO_DINT(Value));
AddUsint := THIS^;
END_METHOD

METHOD PUBLIC AddWord : I_Serializer
VAR_INPUT
	Value : WORD;
END_VAR
jsonSaxWriter.AddUDint(WORD_TO_UDINT(Value));
AddWord := THIS^;
END_METHOD

METHOD PUBLIC Clone : I_Serializer
VAR
	pClone : POINTER TO MockJsonSerializer;
	jsonSize : UDINT;
	pJsonString : POINTER TO STRING;
END_VAR
pClone := __NEW(MockJsonSerializer);
Clone := pClone^;

jsonSize := jsonSaxWriter.GetDocumentLength();

IF jsonSize = 0 THEN
	// no further cloning to do. 
	RETURN;
END_IF

pJsonString := __NEW(BYTE, jsonSize);

IF jsonSaxWriter.CopyDocument(pJsonString^, jsonSize) = 0 THEN
	__DELETE(pJsonString);
	RETURN;
END_IF

pClone^.AddRawJson(pJsonString^);
__DELETE(pJsonString);
END_METHOD

METHOD PUBLIC EndArray : I_Serializer
VAR_INPUT
END_VAR
jsonSaxWriter.EndArray();
EndArray := THIS^;
END_METHOD

METHOD PUBLIC EndObject : I_Serializer
VAR_INPUT
END_VAR
jsonSaxWriter.EndObject();
EndObject := THIS^;
END_METHOD

METHOD FB_exit : BOOL
VAR_INPUT
	bInCopyCode : BOOL; // if TRUE, the exit method is called for exiting an instance that is copied afterwards (online change).
END_VAR
IF bInCopyCode THEN
	RETURN;
END_IF

jsonSaxWriter.ResetDocument();
END_METHOD

METHOD PUBLIC GetSerializedDataLength : UDINT
VAR_INPUT
END_VAR
GetSerializedDataLength := jsonSaxWriter.GetDocumentLength();
END_METHOD

METHOD PUBLIC Reset
VAR_INPUT
END_VAR
jsonSaxWriter.ResetDocument();
END_METHOD

METHOD PUBLIC StartArray : I_Serializer
VAR_INPUT
END_VAR
jsonSaxWriter.StartArray();
StartArray := THIS^;
END_METHOD

METHOD PUBLIC StartObject : I_Serializer
VAR_INPUT
END_VAR
jsonSaxWriter.StartObject();
StartObject := THIS^;
END_METHOD

METHOD TryCopySerializedData : BOOL
VAR_INPUT
	DestinationAddress : PVOID;
	DestinationSize : UDINT;
END_VAR
VAR
	pString : POINTER TO STRING;
END_VAR
pString := DestinationAddress;
TryCopySerializedData := jsonSaxWriter.CopyDocument(pString^, DestinationSize) > 0;
END_METHOD

METHOD TryGetSerializedData : BOOL
VAR_INPUT
	DestinationAddress : PVOID;
	DestinationSize : UDINT;
END_VAR
VAR
	pString : POINTER TO STRING;
END_VAR
pString := DestinationAddress;

IF jsonSaxWriter.CopyDocument(pString^, DestinationSize) = 0 THEN
	RETURN;
END_IF

jsonSaxWriter.ResetDocument();
TryGetSerializedData := TRUE;
END_METHOD

END_FUNCTION_BLOCK

// ---- mobject-deserialization/Tests/DeserializationErrorFactory_TestSuite.TcPOU
FUNCTION_BLOCK DeserializationErrorFactory_TestSuite EXTENDS TcUnit.FB_TestSuite

TestCreateICustomDeserializationFailedError();
TestCreateIncorrectKeyTypeError();
TestCreateIncorrectTypeError();
TestCreateMissingKeyError();
TestCreateInvalidKeyError();

METHOD PUBLIC TestCreateICustomDeserializationFailedError
VAR
	error : CustomDeserializationFailedError('testMessage');
	factory : DeserializationErrorFactory;
	newError : I_Error;
END_VAR
TEST('TestCreateICustomDeserializationFailedError');

newError := factory.CreateCustomDeserializationFailedError('testMessage');

AssertTrue(
	Condition := newError.IsSameAs(error),
	Message := 'Did not produce the correct error type'
);

AssertEquals_String(
	Actual := newError.Message,
	Expected := error.Message,
	Message := 'Did not produce error with correct message'
);

newError.Dispose();

TEST_FINISHED();
END_METHOD

METHOD PUBLIC TestCreateIncorrectKeyTypeError
VAR
	error : IncorrectKeyTypeDeserializationError('testType', 'testKey');
	factory : DeserializationErrorFactory;
	newError : I_Error;
END_VAR
TEST('TestCreateIncorrectKeyTypeError');

newError := factory.CreateIncorrectKeyTypeError('testType','testKey');

AssertTrue(
	Condition := newError.IsSameAs(error),
	Message := 'Did not produce the correct error type'
);

AssertEquals_String(
	Actual := newError.Message,
	Expected := error.Message,
	Message := 'Did not produce error with correct message'
);

newError.Dispose();

TEST_FINISHED();
END_METHOD

METHOD PUBLIC TestCreateIncorrectTypeError
VAR
	error : IncorrectTypeDeserializationError('testType');
	factory : DeserializationErrorFactory;
	newError : I_Error;
END_VAR
TEST('TestCreateIncorrectTypeError');

newError := factory.CreateIncorrectTypeError('testType');

AssertTrue(
	Condition := newError.IsSameAs(error),
	Message := 'Did not produce the correct error type'
);

AssertEquals_String(
	Actual := newError.Message,
	Expected := error.Message,
	Message := 'Did not produce error with correct message'
);

newError.Dispose();

TEST_FINISHED();
END_METHOD

METHOD PUBLIC TestCreateInvalidKeyError
VAR
	error : InvalidKeyDeserializationError;
	factory : DeserializationErrorFactory;
	newError : I_Error;
END_VAR
TEST('TestCreateInvalidKeyError');

newError := factory.CreateInvalidKeyError();

AssertTrue(
	Condition := newError.IsSameAs(error),
	Message := 'Did not produce the correct error type'
);

AssertEquals_String(
	Actual := newError.Message,
	Expected := error.Message,
	Message := 'Did not produce error with correct message'
);

newError.Dispose();

TEST_FINISHED();
END_METHOD

METHOD PUBLIC TestCreateMissingKeyError
VAR
	error : MissingKeyDeserializationError('testKey');
	factory : DeserializationErrorFactory;
	newError : I_Error;
END_VAR
TEST('TestCreateMissingKeyError');

newError := factory.CreateMissingKeyError('testKey');

AssertTrue(
	Condition := newError.IsSameAs(error),
	Message := 'Did not produce the correct error type'
);

AssertEquals_String(
	Actual := newError.Message,
	Expected := error.Message,
	Message := 'Did not produce error with correct message'
);

newError.Dispose();

TEST_FINISHED();
END_METHOD

END_FUNCTION_BLOCK

// ---- mobject-deserialization/Tests/IncorrectKeyTypeDeserializationError_TestSuite.TcPOU
FUNCTION_BLOCK IncorrectKeyTypeDeserializationError_TestSuite EXTENDS TcUnit.FB_TestSuite

TestAccept();
TestErrorType();
TestIsSameAsWithSameErrors();
TestIsSameAsWithDifferentErrors();
TestMessage();
TestSerializeWith();

METHOD PUBLIC TestAccept
VAR
	error : IncorrectKeyTypeDeserializationError('testType', 'testKey');
	visitor : MockErrorVisitor(ExpectedError := error);
END_VAR
TEST('TestAccept');

error.Accept(visitor);

AssertTrue(
	Condition := visitor.VisitedCorrectError,
	Message := 'Did not invoke VisitError on the visitor'
);

TEST_FINISHED();
END_METHOD

METHOD PUBLIC TestErrorType
VAR
	error : IncorrectKeyTypeDeserializationError('testType', 'testKey');
END_VAR
TEST('TestErrorType');

AssertEquals_String(
	Actual := error.ErrorType,
	Expected := 'INCORRECT_DATATYPE_DESERIALIZATION_ERROR',
	Message := 'Did not return the expected ErrorType'
);

TEST_FINISHED();
END_METHOD

METHOD PUBLIC TestIsSameAsWithDifferentErrors
VAR
	error1 : IncorrectKeyTypeDeserializationError('testType', 'testKey');
	error2 : MockError(MockErrorType:='ERROR_TYPE_B',MockMessage:='Message 2');
END_VAR
TEST('TestIsSameAsWithDifferentErrors');

AssertFalse(
	Condition := error1.IsSameAs(error2),
	Message := 'Did not correctly identify errors as being different type'
);

TEST_FINISHED();
END_METHOD

METHOD PUBLIC TestIsSameAsWithSameErrors
VAR
	error1 : IncorrectKeyTypeDeserializationError('testType', 'testKey');
	error2 : MockError(MockErrorType:='INCORRECT_DATATYPE_DESERIALIZATION_ERROR',MockMessage:='Message');
END_VAR
TEST('TestIsSameAsWithSameErrors');

AssertTrue(
	Condition := error1.IsSameAs(error2),
	Message := 'Did not correctly identify errors as being the same type'
);

TEST_FINISHED();
END_METHOD

METHOD PUBLIC TestMessage
VAR
	error : IncorrectKeyTypeDeserializationError('testType', 'testKey');
END_VAR
TEST('TestMessage');

AssertEquals_String(
	Actual := error.Message,
	Expected := 'Deserialization Failed, Incorrect Datatype : testType for key : testKey',
	Message := 'Did not return the expected Message'
);

TEST_FINISHED();
END_METHOD

METHOD PUBLIC TestSerializeWith
VAR
	error : IncorrectKeyTypeDeserializationError('testType', 'testKey');
	serializer : MockJsonSerializer;
	result : T_MAXSTRING;
END_VAR
TEST('TestSerializeWith');

error.SerializeWith(serializer);
serializer.TryGetSerializedData(ADR(result), SIZEOF(result));

AssertEquals_String(
	Actual := result,
	Expected := '{"errorType":"INCORRECT_DATATYPE_DESERIALIZATION_ERROR","message":"Deserialization Failed, Incorrect Datatype : testType for key : testKey"}',
	Message := 'Did not serialize correctly'
);

TEST_FINISHED();
END_METHOD

END_FUNCTION_BLOCK

// ---- mobject-deserialization/Tests/IncorrectTypeDeserializationError_TestSuite.TcPOU
FUNCTION_BLOCK IncorrectTypeDeserializationError_TestSuite EXTENDS TcUnit.FB_TestSuite

TestAccept();
TestErrorType();
TestIsSameAsWithSameErrors();
TestIsSameAsWithDifferentErrors();
TestMessage();
TestSerializeWith();

METHOD PUBLIC TestAccept
VAR
	error : IncorrectTypeDeserializationError('testType');
	visitor : MockErrorVisitor(ExpectedError := error);
END_VAR
TEST('TestAccept');

error.Accept(visitor);

AssertTrue(
	Condition := visitor.VisitedCorrectError,
	Message := 'Did not invoke VisitError on the visitor'
);

TEST_FINISHED();
END_METHOD

METHOD PUBLIC TestErrorType
VAR
	error : IncorrectTypeDeserializationError('testType');
END_VAR
TEST('TestErrorType');

AssertEquals_String(
	Actual := error.ErrorType,
	Expected := 'INCORRECT_DATATYPE_DESERIALIZATION_ERROR',
	Message := 'Did not return the expected ErrorType'
);

TEST_FINISHED();
END_METHOD

METHOD PUBLIC TestIsSameAsWithDifferentErrors
VAR
	error1 : IncorrectTypeDeserializationError('testType');
	error2 : MockError(MockErrorType:='ERROR_TYPE_B',MockMessage:='Message 2');
END_VAR
TEST('TestIsSameAsWithDifferentErrors');

AssertFalse(
	Condition := error1.IsSameAs(error2),
	Message := 'Did not correctly identify errors as being different type'
);

TEST_FINISHED();
END_METHOD

METHOD PUBLIC TestIsSameAsWithSameErrors
VAR
	error1 : IncorrectTypeDeserializationError('testType');
	error2 : MockError(MockErrorType:='INCORRECT_DATATYPE_DESERIALIZATION_ERROR',MockMessage:='Message');
END_VAR
TEST('TestIsSameAsWithSameErrors');

AssertTrue(
	Condition := error1.IsSameAs(error2),
	Message := 'Did not correctly identify errors as being the same type'
);

TEST_FINISHED();
END_METHOD

METHOD PUBLIC TestMessage
VAR
	error : IncorrectTypeDeserializationError('testType');
END_VAR
TEST('TestMessage');

AssertEquals_String(
	Actual := error.Message,
	Expected := 'Deserialization Failed, Incorrect Datatype : testType',
	Message := 'Did not return the expected Message'
);

TEST_FINISHED();
END_METHOD

METHOD PUBLIC TestSerializeWith
VAR
	error : IncorrectTypeDeserializationError('testType');
	serializer : MockJsonSerializer;
	result : T_MAXSTRING;
END_VAR
TEST('TestSerializeWith');

error.SerializeWith(serializer);
serializer.TryGetSerializedData(ADR(result), SIZEOF(result));

AssertEquals_String(
	Actual := result,
	Expected := '{"errorType":"INCORRECT_DATATYPE_DESERIALIZATION_ERROR","message":"Deserialization Failed, Incorrect Datatype : testType"}',
	Message := 'Did not serialize correctly'
);

TEST_FINISHED();
END_METHOD

END_FUNCTION_BLOCK

// ---- mobject-deserialization/Tests/InvalidKeyDeserializationError_TestSuite.TcPOU
FUNCTION_BLOCK InvalidKeyDeserializationError_TestSuite EXTENDS TcUnit.FB_TestSuite

TestAccept();
TestErrorType();
TestIsSameAsWithSameErrors();
TestIsSameAsWithDifferentErrors();
TestMessage();
TestSerializeWith();

METHOD PUBLIC TestAccept
VAR
	error : InvalidKeyDeserializationError;
	visitor : MockErrorVisitor(ExpectedError := error);
END_VAR
TEST('TestAccept');

error.Accept(visitor);

AssertTrue(
	Condition := visitor.VisitedCorrectError,
	Message := 'Did not invoke VisitError on the visitor'
);

TEST_FINISHED();
END_METHOD

METHOD PUBLIC TestErrorType
VAR
	error : InvalidKeyDeserializationError;
END_VAR
TEST('TestErrorType');

AssertEquals_String(
	Actual := error.ErrorType,
	Expected := 'INVALID_KEY_DESERIALIZATION_ERROR',
	Message := 'Did not return the expected ErrorType'
);

TEST_FINISHED();
END_METHOD

METHOD PUBLIC TestIsSameAsWithDifferentErrors
VAR
	error1 : InvalidKeyDeserializationError;
	error2 : MockError(MockErrorType:='ERROR_TYPE_B',MockMessage:='Message 2');
END_VAR
TEST('TestIsSameAsWithDifferentErrors');

AssertFalse(
	Condition := error1.IsSameAs(error2),
	Message := 'Did not correctly identify errors as being different type'
);

TEST_FINISHED();
END_METHOD

METHOD PUBLIC TestIsSameAsWithSameErrors
VAR
	error1 : InvalidKeyDeserializationError;
	error2 : MockError(MockErrorType:='INVALID_KEY_DESERIALIZATION_ERROR',MockMessage:='Message');
END_VAR
TEST('TestIsSameAsWithSameErrors');

AssertTrue(
	Condition := error1.IsSameAs(error2),
	Message := 'Did not correctly identify errors as being the same type'
);

TEST_FINISHED();
END_METHOD

METHOD PUBLIC TestMessage
VAR
	error : InvalidKeyDeserializationError;
END_VAR
TEST('TestMessage');

AssertEquals_String(
	Actual := error.Message,
	Expected := 'Deserialization Failed, Key Cannot Be Empty',
	Message := 'Did not return the expected Message'
);

TEST_FINISHED();
END_METHOD

METHOD PUBLIC TestSerializeWith
VAR
	error : InvalidKeyDeserializationError;
	serializer : MockJsonSerializer;
	result : T_MAXSTRING;
END_VAR
TEST('TestSerializeWith');

error.SerializeWith(serializer);
serializer.TryGetSerializedData(ADR(result), SIZEOF(result));

AssertEquals_String(
	Actual := result,
	Expected := '{"errorType":"INVALID_KEY_DESERIALIZATION_ERROR","message":"Deserialization Failed, Key Cannot Be Empty"}',
	Message := 'Did not serialize correctly'
);

TEST_FINISHED();
END_METHOD

END_FUNCTION_BLOCK

// ---- mobject-deserialization/Tests/Mocks/MockDisposableDeserializer.TcPOU
FUNCTION_BLOCK MockDisposableDeserializer IMPLEMENTS I_Deserializer
VAR
	disposedFlag : BOOL;
END_VAR

METHOD PUBLIC Clone : I_Deserializer
END_METHOD

METHOD PUBLIC Dispose
VAR_INPUT
END_VAR
disposedFlag := TRUE;
END_METHOD

METHOD GetArray : I_Deserializer
VAR_INPUT
END_VAR
END_METHOD

METHOD GetArrayEnumerator : I_DeserializerArrayForwardEnumerator
VAR_INPUT
END_VAR
END_METHOD

METHOD GetElementByIndex : I_Deserializer
VAR_INPUT
	Index : UDINT;
END_VAR
END_METHOD

METHOD GetKeyArray : I_Deserializer
VAR_INPUT
	Key : T_MAXSTRING;
END_VAR
END_METHOD

METHOD GetKeyObject : I_Deserializer
VAR_INPUT
	Key : T_MAXSTRING;
END_VAR
END_METHOD

METHOD GetObject : I_Deserializer
VAR_INPUT
END_VAR
END_METHOD

METHOD GetObjectEnumerator : I_DeserializerObjectForwardEnumerator
VAR_INPUT
END_VAR
END_METHOD

PROPERTY PUBLIC IsDisposed : BOOL
GET
IsDisposed := disposedFlag;
END_GET
END_PROPERTY

METHOD TryDeserializeKeyToObject : BOOL
VAR_INPUT
	Key : T_MAXSTRING;
	Object : I_Deserializable;
	Feedback : I_DeserializerFeedback;
END_VAR
END_METHOD

METHOD TryDeserializeToObject : BOOL
VAR_INPUT
	Object : I_Deserializable;
	Feedback : I_DeserializerFeedback;
END_VAR
END_METHOD

METHOD TryGetBase64 : BOOL
VAR_INPUT
	pBytes : POINTER TO BYTE;
	nBytes : DINT;
	Feedback : I_DeserializerFeedback;
END_VAR
END_METHOD

METHOD TryGetBool : BOOL
VAR_INPUT
	Destination : REFERENCE TO BOOL;
	Feedback : I_DeserializerFeedback;
END_VAR
END_METHOD

METHOD TryGetByte : BOOL
VAR_INPUT
	Destination : REFERENCE TO BYTE;
	Feedback : I_DeserializerFeedback;
END_VAR
END_METHOD

METHOD TryGetDateTime : BOOL
VAR_INPUT
	Destination : REFERENCE TO DATE_AND_TIME;
	Feedback : I_DeserializerFeedback;
END_VAR
END_METHOD

METHOD TryGetDcTime : BOOL
VAR_INPUT
	Destination : REFERENCE TO DCTIME;
	Feedback : I_DeserializerFeedback;
END_VAR
END_METHOD

METHOD TryGetDint : BOOL
VAR_INPUT
	Destination : REFERENCE TO DINT;
	Feedback : I_DeserializerFeedback;
END_VAR
END_METHOD

METHOD TryGetDword : BOOL
VAR_INPUT
	Destination : REFERENCE TO DWORD;
	Feedback : I_DeserializerFeedback;
END_VAR
END_METHOD

METHOD TryGetElementByIndex : BOOL
VAR_INPUT
	Index : UDINT;
	Destination : REFERENCE TO I_Deserializer;
	Feedback : I_DeserializerFeedback;
END_VAR
END_METHOD

METHOD TryGetFileTime : BOOL
VAR_INPUT
	Destination : REFERENCE TO FILETIME;
	Feedback : I_DeserializerFeedback;
END_VAR
END_METHOD

METHOD TryGetHexAsBytes : BOOL
VAR_INPUT
	pBytes : POINTER TO BYTE;
	nBytes : DINT;
	Feedback : I_DeserializerFeedback;
END_VAR
END_METHOD

METHOD TryGetInt : BOOL
VAR_INPUT
	Destination : REFERENCE TO INT;
	Feedback : I_DeserializerFeedback;
END_VAR
END_METHOD

METHOD TryGetKeyBase64 : BOOL
VAR_INPUT
	Key : T_MAXSTRING;
	pBytes : POINTER TO BYTE;
	nBytes : DINT;
	Feedback : I_DeserializerFeedback;
END_VAR
END_METHOD

METHOD TryGetKeyBool : BOOL
VAR_INPUT
	Key : T_MAXSTRING;
	Destination : REFERENCE TO BOOL;
	Feedback : I_DeserializerFeedback;
END_VAR
END_METHOD

METHOD TryGetKeyByte : BOOL
VAR_INPUT
	Key : T_MAXSTRING;
	Destination : REFERENCE TO BYTE;
	Feedback : I_DeserializerFeedback;
END_VAR
END_METHOD

METHOD TryGetKeyDateTime : BOOL
VAR_INPUT
	Key : T_MAXSTRING;
	Destination : REFERENCE TO DATE_AND_TIME;
	Feedback : I_DeserializerFeedback;
END_VAR
END_METHOD

METHOD TryGetKeyDcTime : BOOL
VAR_INPUT
	Key : T_MAXSTRING;
	Destination : REFERENCE TO DCTIME;
	Feedback : I_DeserializerFeedback;
END_VAR
END_METHOD

METHOD TryGetKeyDint : BOOL
VAR_INPUT
	Key : T_MAXSTRING;
	Destination : REFERENCE TO DINT;
	Feedback : I_DeserializerFeedback;
END_VAR
END_METHOD

METHOD TryGetKeyDword : BOOL
VAR_INPUT
	Key : T_MAXSTRING;
	Destination : REFERENCE TO DWORD;
	Feedback : I_DeserializerFeedback;
END_VAR
END_METHOD

METHOD TryGetKeyFileTime : BOOL
VAR_INPUT
	Key : T_MAXSTRING;
	Destination : REFERENCE TO FILETIME;
	Feedback : I_DeserializerFeedback;
END_VAR
END_METHOD

METHOD TryGetKeyHexAsBytes : BOOL
VAR_INPUT
	Key : T_MAXSTRING;
	pBytes : POINTER TO BYTE;
	nBytes : DINT;
	Feedback : I_DeserializerFeedback;
END_VAR
END_METHOD

METHOD TryGetKeyInt : BOOL
VAR_INPUT
	Key : T_MAXSTRING;
	Destination : REFERENCE TO INT;
	Feedback : I_DeserializerFeedback;
END_VAR
END_METHOD

METHOD TryGetKeyLint : BOOL
VAR_INPUT
	Key : T_MAXSTRING;
	Destination : REFERENCE TO LINT;
	Feedback : I_DeserializerFeedback;
END_VAR
END_METHOD

METHOD TryGetKeyLreal : BOOL
VAR_INPUT
	Key : T_MAXSTRING;
	Destination : REFERENCE TO LREAL;
	Feedback : I_DeserializerFeedback;
END_VAR
END_METHOD

METHOD TryGetKeyLtime : BOOL
VAR_INPUT
	Key : T_MAXSTRING;
	Destination : REFERENCE TO LTIME;
	Feedback : I_DeserializerFeedback;
END_VAR
END_METHOD

METHOD TryGetKeyLword : BOOL
VAR_INPUT
	Key : T_MAXSTRING;
	Destination : REFERENCE TO LWORD;
	Feedback : I_DeserializerFeedback;
END_VAR
END_METHOD

METHOD TryGetKeyReal : BOOL
VAR_INPUT
	Key : T_MAXSTRING;
	Destination : REFERENCE TO REAL;
	Feedback : I_DeserializerFeedback;
END_VAR
END_METHOD

METHOD TryGetKeySint : BOOL
VAR_INPUT
	Key : T_MAXSTRING;
	Destination : REFERENCE TO SINT;
	Feedback : I_DeserializerFeedback;
END_VAR
END_METHOD

METHOD TryGetKeyString : BOOL
VAR_INPUT
	Key : T_MAXSTRING;
	Destination : REFERENCE TO T_MAXSTRING;
	Feedback : I_DeserializerFeedback;
END_VAR
END_METHOD

METHOD TryGetKeyStringEx : BOOL
VAR_INPUT
	Key : T_MAXSTRING;
	DestinationAddress : POINTER TO STRING;
	DestinationSize : UDINT;
	Feedback : I_DeserializerFeedback;
END_VAR
END_METHOD

METHOD TryGetKeyTime : BOOL
VAR_INPUT
	Key : T_MAXSTRING;
	Destination : REFERENCE TO TIME;
	Feedback : I_DeserializerFeedback;
END_VAR
END_METHOD

METHOD TryGetKeyTod : BOOL
VAR_INPUT
	Key : T_MAXSTRING;
	Destination : REFERENCE TO TOD;
	Feedback : I_DeserializerFeedback;
END_VAR
END_METHOD

METHOD TryGetKeyUdint : BOOL
VAR_INPUT
	Key : T_MAXSTRING;
	Destination : REFERENCE TO UDINT;
	Feedback : I_DeserializerFeedback;
END_VAR
END_METHOD

METHOD TryGetKeyUint : BOOL
VAR_INPUT
	Key : T_MAXSTRING;
	Destination : REFERENCE TO UINT;
	Feedback : I_DeserializerFeedback;
END_VAR
END_METHOD

METHOD TryGetKeyUlint : BOOL
VAR_INPUT
	Key : T_MAXSTRING;
	Destination : REFERENCE TO ULINT;
	Feedback : I_DeserializerFeedback;
END_VAR
END_METHOD

METHOD TryGetKeyUsint : BOOL
VAR_INPUT
	Key : T_MAXSTRING;
	Destination : REFERENCE TO USINT;
	Feedback : I_DeserializerFeedback;
END_VAR
END_METHOD

METHOD TryGetKeyWord : BOOL
VAR_INPUT
	Key : T_MAXSTRING;
	Destination : REFERENCE TO WORD;
	Feedback : I_DeserializerFeedback;
END_VAR
END_METHOD

METHOD TryGetLint : BOOL
VAR_INPUT
	Destination : REFERENCE TO LINT;
	Feedback : I_DeserializerFeedback;
END_VAR
END_METHOD

METHOD TryGetLreal : BOOL
VAR_INPUT
	Destination : REFERENCE TO LREAL;
	Feedback : I_DeserializerFeedback;
END_VAR
END_METHOD

METHOD TryGetLtime : BOOL
VAR_INPUT
	Destination : REFERENCE TO LTIME;
	Feedback : I_DeserializerFeedback;
END_VAR
END_METHOD

METHOD TryGetLword : BOOL
VAR_INPUT
	Destination : REFERENCE TO LWORD;
	Feedback : I_DeserializerFeedback;
END_VAR
END_METHOD

METHOD TryGetReal : BOOL
VAR_INPUT
	Destination : REFERENCE TO REAL;
	Feedback : I_DeserializerFeedback;
END_VAR
END_METHOD

METHOD TryGetSint : BOOL
VAR_INPUT
	Destination : REFERENCE TO SINT;
	Feedback : I_DeserializerFeedback;
END_VAR
END_METHOD

METHOD TryGetString : BOOL
VAR_INPUT
	Destination : REFERENCE TO T_MAXSTRING;
	Feedback : I_DeserializerFeedback;
END_VAR
END_METHOD

METHOD TryGetStringEx : BOOL
VAR_INPUT
	DestinationAddress : POINTER TO STRING;
	DestinationSize : UDINT;
	Feedback : I_DeserializerFeedback;
END_VAR
END_METHOD

METHOD TryGetTime : BOOL
VAR_INPUT
	Destination : REFERENCE TO TIME;
	Feedback : I_DeserializerFeedback;
END_VAR
END_METHOD

METHOD TryGetTod : BOOL
VAR_INPUT
	Destination : REFERENCE TO TOD;
	Feedback : I_DeserializerFeedback;
END_VAR
END_METHOD

METHOD TryGetUdint : BOOL
VAR_INPUT
	Destination : REFERENCE TO UDINT;
	Feedback : I_DeserializerFeedback;
END_VAR
END_METHOD

METHOD TryGetUint : BOOL
VAR_INPUT
	Destination : REFERENCE TO UINT;
	Feedback : I_DeserializerFeedback;
END_VAR
END_METHOD

METHOD TryGetUlint : BOOL
VAR_INPUT
	Destination : REFERENCE TO ULINT;
	Feedback : I_DeserializerFeedback;
END_VAR
END_METHOD

METHOD TryGetUsint : BOOL
VAR_INPUT
	Destination : REFERENCE TO USINT;
	Feedback : I_DeserializerFeedback;
END_VAR
END_METHOD

METHOD TryGetWord : BOOL
VAR_INPUT
	Destination : REFERENCE TO WORD;
	Feedback : I_DeserializerFeedback;
END_VAR
END_METHOD

END_FUNCTION_BLOCK
